FUNCTION_BLOCK Aguila IMPLEMENTS I_AveVoladora
VAR_INPUT
    velocidad : REAL;
    alturaMaxima : REAL;
END_VAR
VAR
END_VAR


METHOD Volar : BOOL
Volar:= TRUE;
END_METHOD

END_FUNCTION_BLOCK

(* stored: Version 1.1.0.1, ProductVersion 3.1.4024.12
   POU Aguila: Id {6910a7ef-35b8-4bab-b02d-061ddfbf462e}, SpecialFunc None
   Method Volar: Id {9c75935f-3c28-41cb-8df6-ec6b0de9ffab} *)
